PROGRAM INTERNAL P_Example_Array_List
VAR
	eState 		: (IDLE, INSERT, REVERSE, RESIZE, GET, SET, FIND, CLEAR, ADD_FRONT, ADD_BACK, REMOVE, REMOVE_AT);
	fbArray_List: FB_Array_List(2);
	nFind 		: T_Capacity;
	sData 		: WSTRING;
	sRTNData	: ARRAY[0..6] OF WSTRING;
	nCount 		: T_Capacity;
	stError 	: ST_ERROR;
	bSuccess 	: BOOL;
END_VAR

stError := fbArray_List._Error_Status;
CASE eState OF
	INSERT:
		sData := "Cats";	fbArray_List.Insert(sData, 0);
		sData := "Dogs";	fbArray_List.Insert(sData, 1);
		sData := "Ravens";	fbArray_List.Insert(sData, 2);
		sData := "Mollies";	fbArray_List.Insert(sData, 3);
	REVERSE:
		fbArray_List.Reverse();
	RESIZE:
		fbArray_List.Resize(3);
	GET: 
		Scrub();
		fbArray_List
			.Get(sRTNData[0], 0)
			.Get(sRTNData[1], 1)
			.Get(sRTNData[2], 2)
			.Get(sRTNData[3], 3)
			.Get(sRTNData[4], 4)
			.Get(sRTNData[5], 5)
			.Get(sRTNData[6], 6);
	SET:
		sData := "Ravens";	fbArray_List.Set(sData, 0);
		sData := "Mollies";	fbArray_List.Set(sData, 1);
		sData := "Dogs";	fbArray_List.Set(sData, 2);
		sData := "Cats";	fbArray_List.Set(sData, 3);
	FIND:
		sData := "Dogs"; fbArray_List.Find(sData, nIndex => nFind);
	CLEAR:
		fbArray_List.Clear();
	ADD_FRONT:
		sData := "Pythons";fbArray_List.Add_Front(sData);
	ADD_BACK:
		sData := "Anacondas"; fbArray_List.Add_Back(sData);
	REMOVE:
		fbArray_List.Remove(bSuccess => bSuccess);
	REMOVE_AT:
		fbArray_List.Remove_At(2);
		
END_CASE
nCount := fbArray_List._Count;
eState := IDLE;

METHOD PRIVATE Scrub
VAR
	i 			: T_Capacity;
END_VAR
FOR i := 0 TO SIZEOF(sRTNData)/SIZEOF(sRTNData[0])-1 DO sRTNData[i] := ""; END_FOR
END_METHOD

END_PROGRAM

(* stored: Version 1.1.0.1, ProductVersion 3.1.4024.4
   POU P_Example_Array_List: Id {969256da-a7e7-43a9-8f8a-e825c77e7067}, SpecialFunc None
   Method Scrub: Id {082a4892-891e-4a52-937b-41fb028c15e4} *)
